TYPE ST_AbstractLightSource_Status :
STRUCT
	Enabled   : BOOL;
	Error     : BOOL;
	ErrorCode : BYTE;
END_STRUCT
END_TYPE

(* stored: Version 1.1.0.1, ProductVersion 3.1.4026.19
   DUT ST_AbstractLightSource_Status: Id {d8b2a78e-9d39-4531-a629-108178af39d7} *)
